{attribute 'qualified_only'}
VAR_GLOBAL
	Robot1	:	TcoAbbRobotics.TcoIrc5_IO_v_1_x_x;
	Robot2	:	TcoAbbRobotics.TcoOmnicore_IO_v_1_x_x;
END_VAR

(* stored: Version 1.1.0.1, ProductVersion 3.1.4024.12
   GVL GVL: Id {9629ef91-2416-06ad-2c95-b050e672e19e} *)
